Universal Robots PolyScope program: p2_Group1_v2.urp

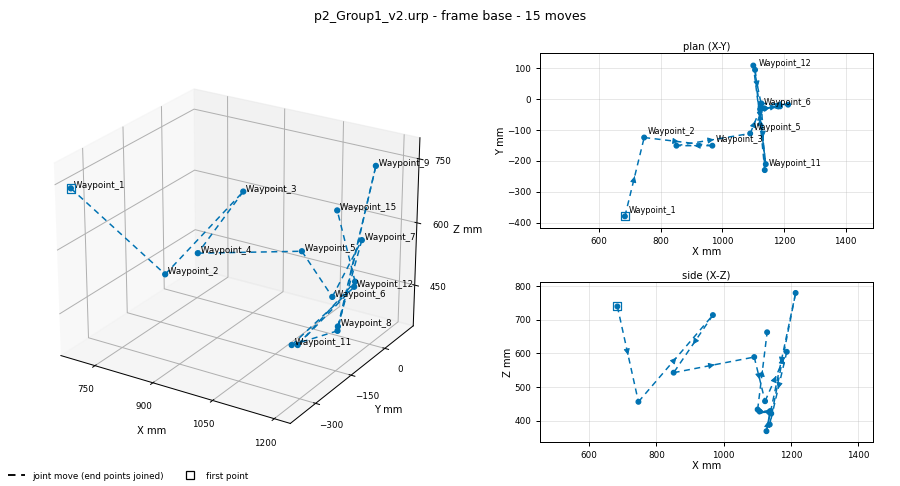
[picture p0: tool path of p2_Group1_v2.urp in frame base, 15 of 15 moves have a stored position in this frame; points joined in program order, loops and branches not executed]
Program p2_Group1_v2 (installation=default directory=/programs/usbdisk/Project2_v2 createdIn=5.13.0 lastSavedIn=5.13.0 robotSerialNumber=20225201357)
Calibrated DH parameters: a=[-0.000097, -0.065329, -0.560646, 0.000001, -0.00004, 0]; d=[0.180831, -263.113709, 285.24385, -21.955837, 0.119737, 0.115719]; alpha=[1.571643, -0.002312, 0.004975, 1.569542, -1.570894, 0]; deltaTheta=[0, 1.463798, 5.013296, -0.193909, 0, 0]
InitVariablesNode
Robot Program (runOnlyOnce=false)
  robotState := read_port_register(200)
  If robotState≟0
    MoveJ speed 60 deg/s, acceleration 80 deg/s^2 (useActiveTCP=true) feature=Base
      Waypoint Waypoint_1: TCP in base x=684.352 y=-379.598 z=739.481 mm, rx=-0.9398 ry=-0.6183 rz=-0.6341 rad; joints [13.89, -75.816, -110.145, -36.067, 15.21, 98.535] deg; TCP offset x=-0.19 y=3.58 z=256.26 mm, rx=0.0015 ry=-2.7841 rz=0 rad
      Waypoint Waypoint_2: TCP in base x=746.846 y=-124.028 z=456.485 mm, rx=-0.2319 ry=-0.2138 rz=-0.0426 rad; joints [13.884, -75.882, -111.557, -52.901, 70.137, 98.537] deg
      Waypoint Waypoint_3: TCP in base x=967.893 y=-150.469 z=713.874 mm, rx=-0.4943 ry=-0.5455 rz=-0.0097 rad; joints [13.782, -91.413, -86.418, -40.865, 56.65, 82.342] deg
      Waypoint Waypoint_4: TCP in base x=851.421 y=-150.528 z=542.965 mm, rx=-0.2467 ry=-0.9137 rz=-0.0026 rad; joints [9.476, -83.633, -123.345, 10.125, 71.547, 83.071] deg
  ElseIf robotState≟1
    MoveJ speed 60 deg/s, acceleration 80 deg/s^2 (useActiveTCP=true) feature=Base
      Waypoint Waypoint_5: motionParameters(nextMotionTime=0.5); TCP in base x=1090.529 y=-110.997 z=589.299 mm, rx=-1.073 ry=-0.7951 rz=0.8305 rad; joints [7.325, -105.039, -97.501, 10.114, 78.069, 16.594] deg
      Waypoint Waypoint_6: motionParameters(nextMotionTime=0.5); TCP in base x=1122.684 y=-32.279 z=458.238 mm, rx=-0.6172 ry=-0.2797 rz=1.2489 rad; joints [7.406, -111.638, -74.782, -46.825, 89.566, 16.579] deg
      Waypoint Waypoint_7: motionParameters(nextMotionTime=0.5); TCP in base x=1187.141 y=-23.043 z=604.846 mm, rx=-0.8218 ry=-0.6468 rz=1.1085 rad; joints [7.402, -111.656, -74.46, -23.813, 89.568, 16.582] deg
      Waypoint Waypoint_8: motionParameters(nextMotionTime=0.5); TCP in base x=1136.524 y=-29.547 z=389.096 mm, rx=-0.5894 ry=-0.2408 rz=1.2638 rad; joints [7.363, -114.813, -75.819, -45.239, 89.827, 16.584] deg
      Waypoint Waypoint_9: motionParameters(nextMotionTime=0.5); TCP in base x=1213.413 y=-17.587 z=779.575 mm, rx=-1.0379 ry=-1.0725 rz=0.897 rad; joints [7.361, -114.719, -71.047, 3.179, 89.824, 16.587] deg
      Waypoint Waypoint_10: motionParameters(nextMotionTime=0.5); TCP in base x=1126.826 y=-13.396 z=369.237 mm, rx=-0.5064 ry=-0.2687 rz=1.2921 rad; joints [6.568, -115.166, -76.733, -45.284, 94.88, 16.585] deg
      Waypoint Waypoint_11: motionParameters(nextMotionTime=0.5); TCP in base x=1137.746 y=-229.721 z=428.842 mm, rx=-0.9448 ry=0.0307 rz=1.0134 rad; joints [5.497, -115.176, -75.039, -44.582, 63.854, 16.585] deg
      Waypoint Waypoint_12: motionParameters(nextMotionTime=0.5); TCP in base x=1106.275 y=95.402 z=427.922 mm, rx=-0.2283 ry=-0.5219 rz=1.3991 rad; joints [5.5, -115.173, -75.012, -44.584, 115.932, 16.607] deg
      Waypoint Waypoint_13: motionParameters(nextMotionTime=0.5); TCP in base x=1141.079 y=-210.411 z=421.597 mm, rx=-0.9031 ry=-0.0044 rz=1.0418 rad; joints [5.477, -115.198, -75.011, -44.582, 67.121, 16.604] deg
      Waypoint Waypoint_14: motionParameters(nextMotionTime=0.5); TCP in base x=1100.661 y=109.384 z=433.595 mm, rx=-0.1904 ry=-0.548 rz=1.4134 rad; joints [5.488, -115.199, -75.01, -44.58, 118.476, 16.603] deg
      Waypoint Waypoint_15: motionParameters(nextMotionTime=0.5); TCP in base x=1128.841 y=-28.909 z=662.855 mm, rx=-0.5926 ry=-0.4121 rz=1.2358 rad; joints [5.659, -111.619, -57.342, -58.965, 95.221, 16.604] deg
